INTERFACE ITF_ControlE_TE2_HMI EXTENDS ITF_BaseControlElement_HMI

METHOD LinkControlEData : BOOL
VAR_INPUT
	stData				: REFERENCE TO ST_ControlE_TE2_HMI_Link;
END_VAR
END_METHOD

END_INTERFACE

(* stored: Version 1.1.0.1, ProductVersion 3.1.4024.15
   Itf ITF_ControlE_TE2_HMI: Id {ca02e696-403f-4957-be76-9caa8cd3fc3f}
   Method LinkControlEData: Id {92d66c81-9f42-4fa1-80f6-1171121a3302} *)
